INTERFACE I_ManualMode EXTENDS I_PackMLMode

END_INTERFACE

(* stored: Version 1.1.0.1, ProductVersion 3.1.4024.12
   Itf I_ManualMode: Id {eb90698e-8345-4db3-9da5-eb1783d425dd} *)
